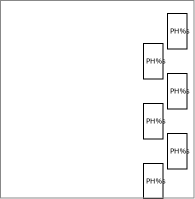
VISUALIZATION _VISU_edit  // 195x199
    Rectangle (167,13 20x36)
        toggle mInst._pPh[7]^._pAdsIf^.bI_Enable
    Rectangle (159,21 36x20), angle 270, "PH%s", tooltip "%S", text variable: mInst._pPh[7]^._lIdx
        p4168582468: mInst._pPh[7]^._pAdsIf^.aO_Name
    Rectangle (167,73 20x36)
        toggle mInst._pPh[8]^._pAdsIf^.bI_Enable
    Rectangle (167,133 20x36)
        toggle mInst._pPh[9]^._pAdsIf^.bI_Enable
    Rectangle (143,43 20x36)
        toggle mInst._pPh[10]^._pAdsIf^.bI_Enable
    Rectangle (143,103 20x36)
        toggle mInst.__pPh[11]^._pAdsIf^.bI_Enable
    Rectangle (143,163 20x36)
        toggle mInst._p_pPh[12]^._pAdsIf^.bI_Enable
    Rectangle (159,81 36x20), angle 270, "PH%s", tooltip "%S", text variable: mInst._pPh[8]^._lIdx
        p4168582468: mInst._pPh[8]^._pAdsIf^.aO_Name
    Rectangle (159,141 36x20), angle 270, "PH%s", tooltip "%S", text variable: mInst._pPh[9]^._lIdx
        p4168582468: mInst._pPh[9]^._pAdsIf^.aO_Name
    Rectangle (135,51 36x20), angle 270, "PH%s", tooltip "%S", text variable: mInst._pPh[10]^._lIdx
        p4168582468: mInst._pPh[10]^._pAdsIf^.aO_Name
    Rectangle (135,111 36x20), angle 270, "PH%s", tooltip "%S", text variable: mInst.__pPh[11]^._lIdx
        p4168582468: mInst.__pPh[11]^._pAdsIf^.aO_Name
    Rectangle (135,171 36x20), angle 270, "PH%s", tooltip "%S", text variable: mInst._p_pPh[12]^._lIdx
        p4168582468: mInst._p_pPh[12]^._pAdsIf^.aO_Name
END_VISUALIZATION

(* stored: Version 1.1.0.1, ProductVersion 3.1.4024.11
   Visu _VISU_edit: Id {dea2f20a-1378-42e5-9bba-0c0fb224265b} *)
